FUNCTION DEG_TO_RAD : LREAL
VAR_INPUT
    degrees : LREAL;
END_VAR
VAR
END_VAR

DEG_TO_RAD := degrees / 180.0 * PI;

END_FUNCTION

(* stored: Version 1.1.0.1, ProductVersion 3.1.4018.5
   POU DEG_TO_RAD: Id {633938d1-ee6d-45ac-aed6-d1f11529bcff}, SpecialFunc None *)
